VAR_GLOBAL
    // Disconnector 1 IO Structure
    stDisconnector1_IO: ST_DisconnectorIO;
    
    // Contactor 1 IO Structure  
    stContactor1_IO: ST_ContactorIO;
	
    // IO Structure
    stCircuitBreaker1_IO: ST_CircuitBreakerIO;	
END_VAR

(* stored: Version 1.1.0.1, ProductVersion 3.1.4024.15
   GVL GVL_IO: Id {a3bfcdbb-eddf-4706-a021-5158f869c8d3} *)
